PROGRAM PRG_FB_ALARM_LogTableManual
VAR

	fbALARM_LogTable		: ALARMS.FB_ALARM_LogTable;
	
	bResetActive			: BOOL;
	//IN_OUT variables

	stAlarmTable			:	ST_AlarmsTable;
	aAlarms 				: 	ARRAY [0..cMAX_ALARM_GROUP] OF ST_Alarms;
	aAlarmsSettings 		: 	ARRAY [0..cMAX_ALARM_GROUP] OF ST_AlarmSettings;
	stCTDateTime			: 	ST_SYSTEM_DateTime;
	
	nI	: INT;

END_VAR

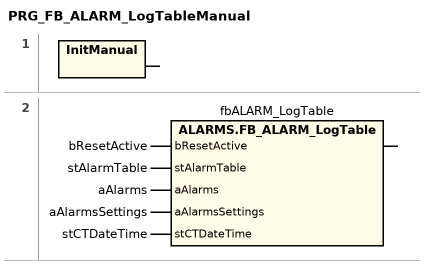
// NETWORK 1
InitManual();

// NETWORK 2
fbALARM_LogTable(
    bResetActive := bResetActive,
    stAlarmTable := stAlarmTable,
    aAlarms := aAlarms,
    aAlarmsSettings := aAlarmsSettings,
    stCTDateTime := stCTDateTime); // ALARMS.FB_ALARM_LogTable

ACTION InitManual:



aAlarms[0].nMessage := 16#00000001;

stCTDateTime.strHMIDateTime := 'Alarm No.';
FOR nI := 0 TO 255 DO	
	stAlarmTable.aMsgAux[nI].sTextMessage := TO_STRING(nI);		
END_FOR
END_ACTION

END_PROGRAM

(* stored: Version 1.1.0.1
   POU PRG_FB_ALARM_LogTableManual: Id {40a84d3c-0d1d-46ca-b11a-27e190de3ddf}, SpecialFunc None
   Action InitManual: Id {af4fa378-0741-4677-b846-ff59ad3bb584} *)
